  MoveL 686 to (188.8, 224.64, -20.05) mm, rotated rx -180 ry 0 rz 179.9 deg; joints [16.387, -39.153, 104.46, -161.937, 65.449, 172.769]
  MoveL 687 to (187.57, 224.64, -20.05) mm, rotated rx 180 ry 0 rz 179.9 deg; joints [16.4, -39.199, 104.569, -161.931, 65.509, 172.785]
  MoveL 688 to (-182.67, 224.64, -20.05) mm, rotated rx 180 ry 0 rz 179.9 deg; joints [21.726, -50.447, 133.658, -158.097, 82.764, 177.685]
  MoveL 689 to (-188.8, 224.64, -20.05) mm, rotated rx 180 ry 0 rz 179.9 deg; joints [21.842, -50.588, 134.091, -157.994, 83.041, 177.782]
  MoveL 690 to (-189.1, 224.63, -20.05) mm, rotated rx 180 ry 0 rz 179.9 deg; joints [21.849, -50.594, 134.112, -157.988, 83.054, 177.787]
  MoveL 691 to (-189.41, 224.59, -20.05) mm, rotated rx 180 ry 0 rz 179.9 deg; joints [21.856, -50.601, 134.133, -157.981, 83.068, 177.792]
  MoveL 692 to (-189.72, 224.54, -20.05) mm, rotated rx 180 ry 0 rz 179.9 deg; joints [21.864, -50.608, 134.153, -157.973, 83.081, 177.796]
  MoveL 693 to (-190.02, 224.47, -20.05) mm, rotated rx 180 ry 0 rz 179.9 deg; joints [21.874, -50.614, 134.173, -157.965, 83.093, 177.8]
  MoveL 694 to (-190.28, 224.39, -20.05) mm, rotated rx 180 ry 0 rz 179.9 deg; joints [21.882, -50.619, 134.188, -157.957, 83.103, 177.803]
  MoveL 695 to (-190.53, 224.3, -20.05) mm, rotated rx 180 ry 0 rz 179.9 deg; joints [21.891, -50.624, 134.204, -157.948, 83.113, 177.806]
  MoveL 696 to (-190.78, 224.2, -20.05) mm, rotated rx -180 ry 0 rz 179.9 deg; joints [21.901, -50.629, 134.219, -157.939, 83.123, 177.809]
  MoveL 697 to (-191.03, 224.08, -20.05) mm, rotated rx 180 ry 0 rz 179.9 deg; joints [21.911, -50.634, 134.233, -157.928, 83.132, 177.811]
  MoveL 698 to (-191.28, 223.93, -20.05) mm, rotated rx 180 ry 0 rz 179.9 deg; joints [21.923, -50.638, 134.247, -157.917, 83.141, 177.814]
  MoveL 699 to (-191.54, 223.77, -20.05) mm, rotated rx 180 ry 0 rz 179.9 deg; joints [21.935, -50.643, 134.26, -157.905, 83.15, 177.816]
  MoveL 700 to (-191.79, 223.59, -20.05) mm, rotated rx 180 ry 0 rz 179.9 deg; joints [21.949, -50.647, 134.272, -157.892, 83.158, 177.818]
  MoveL 701 to (-192.04, 223.38, -20.05) mm, rotated rx 180 ry 0 rz 179.9 deg; joints [21.964, -50.651, 134.284, -157.878, 83.166, 177.819]
  MoveL 702 to (-192.27, 223.16, -20.05) mm, rotated rx 180 ry 0 rz 179.9 deg; joints [21.978, -50.654, 134.294, -157.863, 83.173, 177.82]
  MoveL 703 to (-192.48, 222.94, -20.05) mm, rotated rx -180 ry 0 rz 179.9 deg; joints [21.992, -50.657, 134.302, -157.849, 83.179, 177.821]
  MoveL 704 to (-192.68, 222.69, -20.05) mm, rotated rx -180 ry 0 rz 179.9 deg; joints [22.008, -50.659, 134.31, -157.833, 83.184, 177.821]
  MoveL 705 to (-192.86, 222.44, -20.05) mm, rotated rx 180 ry 0 rz 179.9 deg; joints [22.024, -50.661, 134.315, -157.818, 83.188, 177.821]
  MoveL 706 to (-193.02, 222.19, -20.05) mm, rotated rx 180 ry 0 rz 179.9 deg; joints [22.039, -50.663, 134.32, -157.803, 83.191, 177.82]
  MoveL 707 to (-193.16, 221.93, -20.05) mm, rotated rx -180 ry 0 rz 179.9 deg; joints [22.053, -50.664, 134.322, -157.788, 83.193, 177.819]
  MoveL 708 to (-193.29, 221.68, -20.05) mm, rotated rx 180 ry 0 rz 179.9 deg; joints [22.068, -50.665, 134.323, -157.774, 83.194, 177.818]
  MoveL 709 to (-193.39, 221.43, -20.05) mm, rotated rx 180 ry 0 rz 179.9 deg; joints [22.082, -50.665, 134.324, -157.76, 83.195, 177.816]
  MoveL 710 to (-193.48, 221.18, -20.05) mm, rotated rx 180 ry 0 rz 179.9 deg; joints [22.095, -50.665, 134.323, -157.746, 83.195, 177.815]
  MoveL 711 to (-193.55, 220.92, -20.05) mm, rotated rx 180 ry 0 rz 179.9 deg; joints [22.109, -50.664, 134.321, -157.733, 83.194, 177.813]
  MoveL 712 to (-193.62, 220.62, -20.05) mm, rotated rx 180 ry 0 rz 179.9 deg; joints [22.124, -50.663, 134.317, -157.717, 83.192, 177.81]
  MoveL 713 to (-193.68, 220.31, -20.05) mm, rotated rx -180 ry 0 rz 179.9 deg; joints [22.14, -50.662, 134.312, -157.701, 83.189, 177.807]
  MoveL 714 to (-193.71, 220, -20.05) mm, rotated rx 180 ry 0 rz 179.9 deg; joints [22.155, -50.66, 134.305, -157.685, 83.185, 177.804]
  MoveL 715 to (-193.72, 219.7, -20.05) mm, rotated rx -180 ry 0 rz 179.9 deg; joints [22.17, -50.658, 134.297, -157.67, 83.181, 177.8]
  MoveL 716 to (-193.72, 216.02, -20.05) mm, rotated rx 180 ry 0 rz 179.9 deg; joints [22.343, -50.626, 134.191, -157.492, 83.119, 177.753]
  MoveL 717 to (-193.72, 215.4, -20.05) mm, rotated rx 180 ry 0 rz 179.9 deg; joints [22.372, -50.621, 134.174, -157.463, 83.109, 177.745]
  MoveL 718 to (-193.7, 215.09, -20.05) mm, rotated rx -180 ry 0 rz 179.9 deg; joints [22.386, -50.618, 134.164, -157.448, 83.103, 177.741]
  MoveL 719 to (-193.67, 214.79, -20.05) mm, rotated rx -180 ry 0 rz 179.9 deg; joints [22.4, -50.615, 134.152, -157.434, 83.096, 177.737]
  MoveL 720 to (-192.48, 207.26, -20.05) mm, rotated rx -180 ry 0 rz 179.9 deg; joints [22.73, -50.523, 133.848, -157.092, 82.916, 177.619]
  MoveL 721 to (-126.84, -206.97, -20.05) mm, rotated rx 180 ry 0 rz 179.9 deg; joints [37.506, -42.708, 112.246, -140.464, 72.99, 167.352]
  MoveL 722 to (-126.77, -207.43, -20.05) mm, rotated rx 180 ry 0 rz 179.9 deg; joints [37.519, -42.697, 112.217, -140.447, 72.979, 167.337]
  MoveC 723 to (-127, -208.24, -20.05) mm, rotated rx 180 ry 0 rz 179.9 deg; joints [37.552, -42.686, 112.19, -140.411, 72.974, 167.317] to (-127.77, -208.59, -20.05) mm, rotated rx -180 ry 0 rz 179.9 deg; joints [37.582, -42.701, 112.225, -140.384, 72.996, 167.322]
  MoveL 724 to (-132.34, -208.5, -20.05) mm, rotated rx 180 ry 0 rz 179.9 deg; joints [37.694, -42.834, 112.543, -140.306, 73.164, 167.415]
  MoveC 725 to (-133.05, -208.49, -19.76) mm, rotated rx -180 ry 0 rz 179.9 deg; joints [37.711, -42.871, 112.596, -140.291, 73.179, 167.42] to (-133.34, -208.48, -19.05) mm, rotated rx 180 ry 0 rz 179.9 deg; joints [37.718, -42.922, 112.624, -140.28, 73.164, 167.403]
  Set speed (1000.0 mm/s)
  MoveL 726 to (-133.34, -208.48, 15) mm, rotated rx 180 ry 0 rz 179.9 deg; joints [37.7, -44.922, 112.94, -139.958, 71.867, 166.276]
  MoveL 727 to (-133.34, -208.48, 15) mm, rotated rx 180 ry 0 rz 179.9 deg; joints [37.7, -44.922, 112.94, -139.958, 71.867, 166.276]
